{attribute 'qualified_only'}
VAR_GLOBAL
	bBool1 : BOOL := FALSE;
	bBool2 : BOOL := TRUE;
END_VAR

(* stored: Version 1.1.0.1, ProductVersion 3.1.4024.12
   GVL Globals: Id {1f9bb3f1-bbc7-4e7f-9953-11c512179d55} *)
